// TIA Portal V20 export
FUNCTION_BLOCK "LER_EQP_Interface"   // FB62, LAD
// stored: Access Published, MemoryReserve 100, SetENOAutomatically false
   VAR_INPUT
      enable : Bool;
      executeCmd : Bool;
      clock : Bool;
      heartBeat : Byte;
      unitStatus : "LAF_typeUnitStatus";
      unitAlarms : "LAF_typeAlarms";
      otherStationStatus : "LER_typeCommunicationUnitStatusRCV";
      partData : "LER_typePartData";
   END_VAR
   VAR_OUTPUT
      error : Bool;
      status : Word;
   END_VAR
   VAR_IN_OUT
      StackCommunication : "LER_typeCommunication";
      configuration : "LER_typeCommunicationConfiguration";
      moduleInterface : "LER_typeCommunicationInterface";
      controlNode : "LER_typeCommunicationControlNode";
   END_VAR
   VAR
      instEQP_Interface_Communication : "LER_EQP_Communication";
      statStkHeartBeat : Byte;
      statStackState : Struct
         Stop : Bool;
         Abort : Bool;
         Hold : Bool;
         Complete : Bool;
         Idle : Bool;
         TotalStop : Bool;
      END_STRUCT;
      statTonTimer : Array[0..9] of TON_TIME;
      statTofTimer : Array[0..9] of TOF_TIME;
   END_VAR
   VAR CONSTANT
      STATUS_NO_ERROR_OCCURRED : Word := 16#0;
      ERR_HEARTBEAT_ERROR : Word := 16#8000;
   END_VAR
BEGIN

REGION Network 1: EQP Interface Stack State
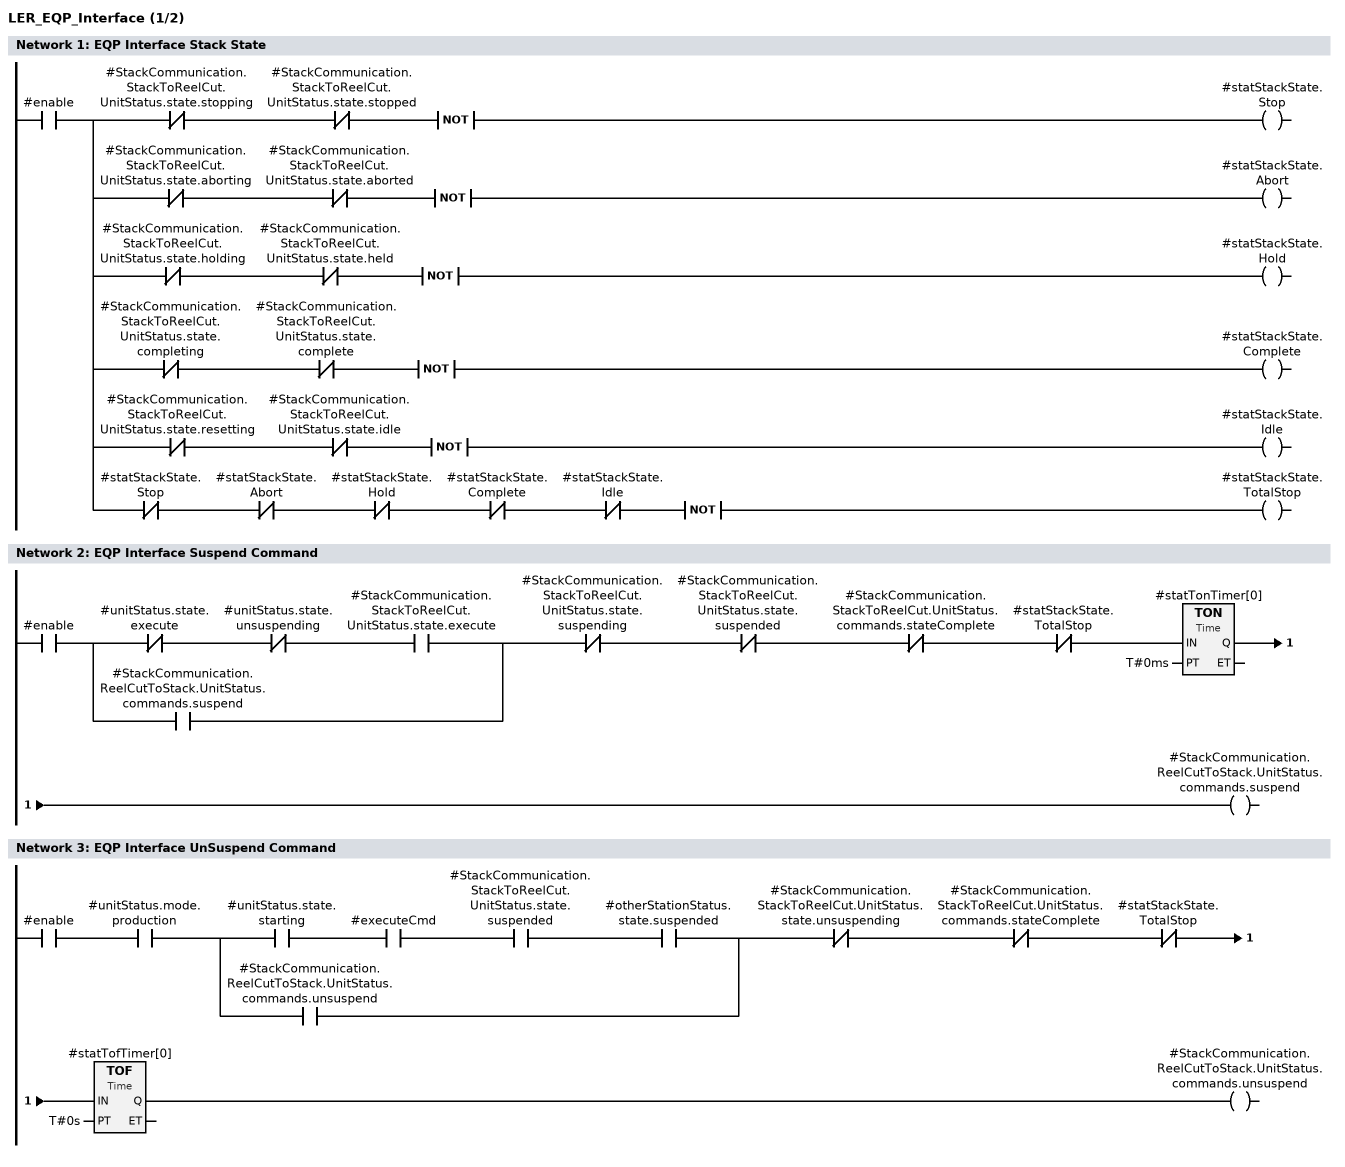
   RUNG wire#powerrail
      Contact( #enable )
      wire#w1
      I_Contact( #StackCommunication.StackToReelCut.UnitStatus.state.stopping )
      I_Contact( #StackCommunication.StackToReelCut.UnitStatus.state.stopped )
      Not()
      Coil( #statStackState.Stop )
   END_RUNG
   RUNG wire#w1
      I_Contact( #StackCommunication.StackToReelCut.UnitStatus.state.aborting )
      I_Contact( #StackCommunication.StackToReelCut.UnitStatus.state.aborted )
      Not()
      Coil( #statStackState.Abort )
   END_RUNG
   RUNG wire#w1
      I_Contact( #StackCommunication.StackToReelCut.UnitStatus.state.holding )
      I_Contact( #StackCommunication.StackToReelCut.UnitStatus.state.held )
      Not()
      Coil( #statStackState.Hold )
   END_RUNG
   RUNG wire#w1
      I_Contact( #StackCommunication.StackToReelCut.UnitStatus.state.completing )
      I_Contact( #StackCommunication.StackToReelCut.UnitStatus.state.complete )
      Not()
      Coil( #statStackState.Complete )
   END_RUNG
   RUNG wire#w1
      I_Contact( #StackCommunication.StackToReelCut.UnitStatus.state.resetting )
      I_Contact( #StackCommunication.StackToReelCut.UnitStatus.state.idle )
      Not()
      Coil( #statStackState.Idle )
   END_RUNG
   RUNG wire#w1
      I_Contact( #statStackState.Stop )
      I_Contact( #statStackState.Abort )
      I_Contact( #statStackState.Hold )
      I_Contact( #statStackState.Complete )
      I_Contact( #statStackState.Idle )
      Not()
      Coil( #statStackState.TotalStop )
   END_RUNG
   // the same network as SCL:
   #statStackState.Stop := NOT (#enable AND NOT #StackCommunication.StackToReelCut.UnitStatus.state.stopping AND NOT #StackCommunication.StackToReelCut.UnitStatus.state.stopped);
   #statStackState.Abort := NOT (#enable AND NOT #StackCommunication.StackToReelCut.UnitStatus.state.aborting AND NOT #StackCommunication.StackToReelCut.UnitStatus.state.aborted);
   #statStackState.Hold := NOT (#enable AND NOT #StackCommunication.StackToReelCut.UnitStatus.state.holding AND NOT #StackCommunication.StackToReelCut.UnitStatus.state.held);
   #statStackState.Complete := NOT (#enable AND NOT #StackCommunication.StackToReelCut.UnitStatus.state.completing AND NOT #StackCommunication.StackToReelCut.UnitStatus.state.complete);
   #statStackState.Idle := NOT (#enable AND NOT #StackCommunication.StackToReelCut.UnitStatus.state.resetting AND NOT #StackCommunication.StackToReelCut.UnitStatus.state.idle);
   #statStackState.TotalStop := NOT (#enable AND NOT #statStackState.Stop AND NOT #statStackState.Abort AND NOT #statStackState.Hold AND NOT #statStackState.Complete AND NOT #statStackState.Idle);
END_REGION

REGION Network 2: EQP Interface Suspend Command
   RUNG wire#powerrail
      Contact( #enable )
      wire#w1
      I_Contact( #unitStatus.state.execute )
      I_Contact( #unitStatus.state.unsuspending )
      Contact( #StackCommunication.StackToReelCut.UnitStatus.state.execute )
      wire#w2
      I_Contact( #StackCommunication.StackToReelCut.UnitStatus.state.suspending )
      I_Contact( #StackCommunication.StackToReelCut.UnitStatus.state.suspended )
      I_Contact( #StackCommunication.StackToReelCut.UnitStatus.commands.stateComplete )
      I_Contact( #statStackState.TotalStop )
      { S7_Templates := "time_type := Time" } #statTonTimer[0].TON(pt := T#0ms, et =>)
      Coil( #StackCommunication.ReelCutToStack.UnitStatus.commands.suspend )
   END_RUNG
   RUNG wire#w1
      Contact( #StackCommunication.ReelCutToStack.UnitStatus.commands.suspend )
   END_RUNG wire#w2
   // the same network as SCL:
   #statTonTimer[0].TON(IN := #enable AND ((NOT #unitStatus.state.execute AND NOT #unitStatus.state.unsuspending AND #StackCommunication.StackToReelCut.UnitStatus.state.execute) OR #StackCommunication.ReelCutToStack.UnitStatus.commands.suspend) AND NOT #StackCommunication.StackToReelCut.UnitStatus.state.suspending AND NOT #StackCommunication.StackToReelCut.UnitStatus.state.suspended AND NOT #StackCommunication.StackToReelCut.UnitStatus.commands.stateComplete AND NOT #statStackState.TotalStop,
                        PT := T#0ms);
   #StackCommunication.ReelCutToStack.UnitStatus.commands.suspend := #statTonTimer[0].Q;
END_REGION

REGION Network 3: EQP Interface UnSuspend Command
   RUNG wire#powerrail
      Contact( #enable )
      Contact( #unitStatus.mode.production )
      wire#w1
      Contact( #unitStatus.state.starting )
      Contact( #executeCmd )
      Contact( #StackCommunication.StackToReelCut.UnitStatus.state.suspended )
      Contact( #otherStationStatus.state.suspended )
      wire#w2
      I_Contact( #StackCommunication.StackToReelCut.UnitStatus.state.unsuspending )
      I_Contact( #StackCommunication.StackToReelCut.UnitStatus.commands.stateComplete )
      I_Contact( #statStackState.TotalStop )
      { S7_Templates := "time_type := Time" } #statTofTimer[0].TOF(pt := T#0s, et =>)
      Coil( #StackCommunication.ReelCutToStack.UnitStatus.commands.unsuspend )
   END_RUNG
   RUNG wire#w1
      Contact( #StackCommunication.ReelCutToStack.UnitStatus.commands.unsuspend )
   END_RUNG wire#w2
   // the same network as SCL:
   #statTofTimer[0].TOF(IN := #enable AND #unitStatus.mode.production AND ((#unitStatus.state.starting AND #executeCmd AND #StackCommunication.StackToReelCut.UnitStatus.state.suspended AND #otherStationStatus.state.suspended) OR #StackCommunication.ReelCutToStack.UnitStatus.commands.unsuspend) AND NOT #StackCommunication.StackToReelCut.UnitStatus.state.unsuspending AND NOT #StackCommunication.StackToReelCut.UnitStatus.commands.stateComplete AND NOT #statStackState.TotalStop,
                        PT := T#0s);
   #StackCommunication.ReelCutToStack.UnitStatus.commands.unsuspend := #statTofTimer[0].Q;
END_REGION

REGION Network 4: EQP Interface StateComplete (SC)
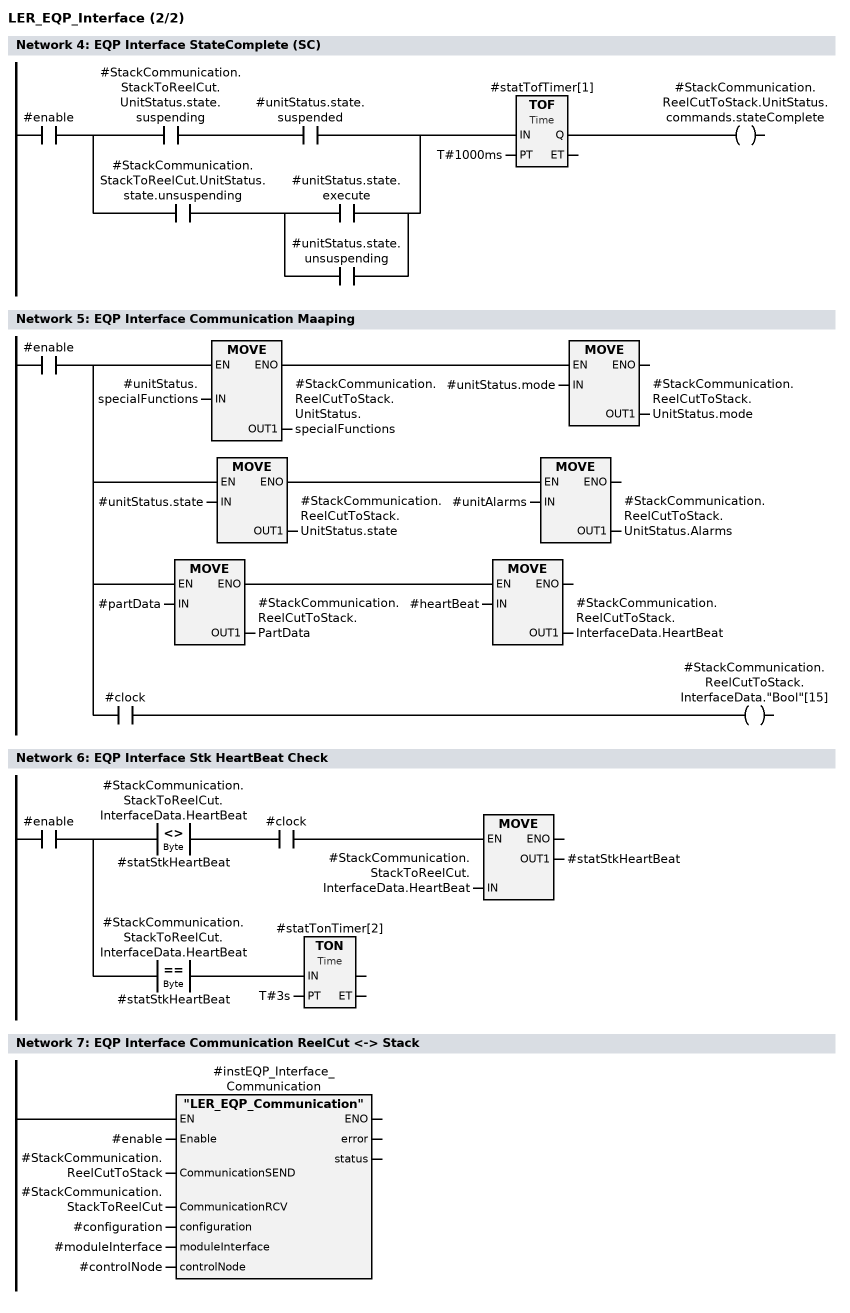
   RUNG wire#powerrail
      Contact( #enable )
      wire#w1
      Contact( #StackCommunication.StackToReelCut.UnitStatus.state.suspending )
      Contact( #unitStatus.state.suspended )
      wire#w2
      { S7_Templates := "time_type := Time" } #statTofTimer[1].TOF(pt := T#1000ms, et =>)
      Coil( #StackCommunication.ReelCutToStack.UnitStatus.commands.stateComplete )
   END_RUNG
   RUNG wire#w1
      Contact( #StackCommunication.StackToReelCut.UnitStatus.state.unsuspending )
      wire#w3
      Contact( #unitStatus.state.execute )
   END_RUNG wire#w2
   RUNG wire#w3
      Contact( #unitStatus.state.unsuspending )
   END_RUNG wire#w2
   // the same network as SCL:
   #statTofTimer[1].TOF(IN := #enable AND ((#StackCommunication.StackToReelCut.UnitStatus.state.suspending AND #unitStatus.state.suspended) OR (#StackCommunication.StackToReelCut.UnitStatus.state.unsuspending AND (#unitStatus.state.execute OR #unitStatus.state.unsuspending))),
                        PT := T#1000ms);
   #StackCommunication.ReelCutToStack.UnitStatus.commands.stateComplete := #statTofTimer[1].Q;
END_REGION

REGION Network 5: EQP Interface Communication Maaping
   RUNG wire#powerrail
      Contact( #enable )
      wire#w1
      Move(in := #unitStatus.specialFunctions, out1 => #StackCommunication.ReelCutToStack.UnitStatus.specialFunctions)
      Move(in := #unitStatus.mode, out1 => #StackCommunication.ReelCutToStack.UnitStatus.mode)
   END_RUNG
   RUNG wire#w1
      Move(in := #unitStatus.state, out1 => #StackCommunication.ReelCutToStack.UnitStatus.state)
      Move(in := #unitAlarms, out1 => #StackCommunication.ReelCutToStack.UnitStatus.Alarms)
   END_RUNG
   RUNG wire#w1
      Move(in := #partData, out1 => #StackCommunication.ReelCutToStack.PartData)
      Move(in := #heartBeat, out1 => #StackCommunication.ReelCutToStack.InterfaceData.HeartBeat)
   END_RUNG
   RUNG wire#w1
      Contact( #clock )
      Coil( #StackCommunication.ReelCutToStack.InterfaceData."Bool"[15] )
   END_RUNG
   // the same network as SCL:
   IF #enable THEN
       #StackCommunication.ReelCutToStack.UnitStatus.specialFunctions := #unitStatus.specialFunctions;
       #StackCommunication.ReelCutToStack.UnitStatus.mode := #unitStatus.mode;
       #StackCommunication.ReelCutToStack.UnitStatus.state := #unitStatus.state;
       #StackCommunication.ReelCutToStack.UnitStatus.Alarms := #unitAlarms;
       #StackCommunication.ReelCutToStack.PartData := #partData;
       #StackCommunication.ReelCutToStack.InterfaceData.HeartBeat := #heartBeat;
   END_IF;
   #StackCommunication.ReelCutToStack.InterfaceData."Bool"[15] := #enable AND #clock;
END_REGION

REGION Network 6: EQP Interface Stk HeartBeat Check
   RUNG wire#powerrail
      Contact( #enable )
      wire#w1
      { S7_Templates := "SrcType := Byte" } NE_Contact(in1 := #StackCommunication.StackToReelCut.InterfaceData.HeartBeat, in2 := #statStkHeartBeat)
      Contact( #clock )
      Move(in := #StackCommunication.StackToReelCut.InterfaceData.HeartBeat, out1 => #statStkHeartBeat)
   END_RUNG
   RUNG wire#w1
      { S7_Templates := "SrcType := Byte" } EQ_Contact(in1 := #StackCommunication.StackToReelCut.InterfaceData.HeartBeat, in2 := #statStkHeartBeat)
      { S7_Templates := "time_type := Time" } #statTonTimer[2].TON(pt := T#3s, et =>)
   END_RUNG
   // the same network as SCL:
   IF #enable AND (#StackCommunication.StackToReelCut.InterfaceData.HeartBeat <> #statStkHeartBeat) AND #clock THEN
       #statStkHeartBeat := #StackCommunication.StackToReelCut.InterfaceData.HeartBeat;
   END_IF;
   #statTonTimer[2].TON(IN := #enable AND (#StackCommunication.StackToReelCut.InterfaceData.HeartBeat = #statStkHeartBeat),
                        PT := T#3s);
END_REGION

REGION Network 7: EQP Interface Communication ReelCut <-> Stack
   RUNG wire#powerrail
      #instEQP_Interface_Communication(Enable := #enable, CommunicationSEND := #StackCommunication.ReelCutToStack, CommunicationRCV := #StackCommunication.StackToReelCut, configuration := #configuration, moduleInterface := #moduleInterface, controlNode := #controlNode, error =>, status =>)
   END_RUNG
   // the same network as SCL:
   #instEQP_Interface_Communication(Enable := #enable,   // "LER_EQP_Communication"
                           CommunicationSEND := #StackCommunication.ReelCutToStack,
                           CommunicationRCV := #StackCommunication.StackToReelCut,
                           configuration := #configuration,
                           moduleInterface := #moduleInterface,
                           controlNode := #controlNode);
END_REGION

REGION Network 8 (SCL): Error Check
   REGION Error Code Search

       IF #enable AND NOT #configuration.disableAlarms THEN
           IF #statTonTimer[2].Q THEN
               #status := #ERR_HEARTBEAT_ERROR;

           ELSIF #instEQP_Interface_Communication.error THEN
               #status := #instEQP_Interface_Communication.status;

           ELSE
               #status := #STATUS_NO_ERROR_OCCURRED;

           END_IF;
       ELSE
           #status := #STATUS_NO_ERROR_OCCURRED;

       END_IF;


       // Error Bit
       #error := #status <> 0;

   END_REGION
END_REGION

REGION Network 9 (SCL): ##### Outputs mapping #####
   #moduleInterface.monitoring.error := #error;
   #moduleInterface.monitoring.status := #status;

   #controlNode.monitoring := #moduleInterface.monitoring;
END_REGION
END_FUNCTION_BLOCK
